// TIA Portal V19 export
VAR_GLOBAL   // PLC tag table "conveyor6m"
   "Belt Conveyor (6m) 0" AT %Q0.4 : Bool;
   "memedge-6m-0" AT %M1.0 : Bool;
   "memedge-6m-1" AT %M1.1 : Bool;
   "memedge-6m-2" AT %M1.2 : Bool;
   "memedge-6m-3" AT %M1.3 : Bool;
   "memedge-6m-4" AT %M1.4 : Bool;
   "memedge-6m-5" AT %M1.5 : Bool;
   "mem-6m-start" AT %M1.6 : Bool;
   "memory-6m-0" AT %M1.7 : Bool;
END_VAR
